//---------------------------------------------------------------------------------------------------------------
//
//  HAUD 2024.11.21
//
//
//  fb_Instance
//  - base class for process instance to work with fb_ProcessCollector
//  - basic check and var names, so you can build your procedures with it
//  - processes are connected via linked list
//
//  - inherit this base class for your application, call Check() cyclic
//
//---------------------------------------------------------------------------------------------------------------//
// This SOFTWARE is provided as an Exemple by THE PROVIDER "as is" and "with all faults." THE PROVIDER makes no  //
// representations or warranties of any kind concerning the safety, suitability, lack of viruses, inaccuracies,  //
// typographical errors, or other harmful components of this SOFTWARE. There are inherent dangers in the use of  //
// any software, and you are solely responsible for determining whether this SOFTWARE is compatible with your    //
// equipment and other software installed on your equipment. You are also solely responsible for the protection  //
// of your equipment and backup of your data, and THE PROVIDER will not be liable for any damages you may suffer //
// in connection with using, modifying, or distributing this SOFTWARE.                                           //
//---------------------------------------------------------------------------------------------------------------//
FUNCTION_BLOCK fb_Instance
VAR
  _eState                 : E_INSTANCE_STATE;  // local state machine for infeed procedure
  _eStateProgress         : E_PROGRESS; // substate for lacal state machine

  _eInit                  : E_PROGRESS;
  _eCheck                 : E_INSTANCE_CHECK;  // pointer checks

  // XTS station range
  _nStationLast           : UINT;
  _nStationFirst          : UINT;

  // process index
  _nProcess               : UINT;

  // local ctrl / state datafields for you to use
  _Ctrl                   : ST_PROCESS_CTRL;   // control to write, connected by reference to _ItfProcessCollector
  _State                  : ST_PROCESS_STATE;  // state   to read,  connected by reference to _ItfProcessCollector

  _ItfProcessCollector    : ARRAY[1..MAX_PROCESS] OF I_ProcessCollector;

  _ItfProcessList         : ARRAY[1..MAX_PROCESS] OF I_Process_LinkedList;  // access to all linked lists for process entry
  _ListResult             : ST_PROCESS_LIST_RESULT;
  _ProcessData            : ST_PROCESS_DATA;

  {attribute 'displaymode':='bin'}
  _wTargetUsed            : T_PROCESS;  // bits use XtsStation in target process
  _wTargetMask            : ARRAY[1..SIZEOF(T_PROCESS)*8] OF BYTE;

  _stMsg                  : ST_Message;
  _MessageLevel           : E_MessageType;
END_VAR

METHOD Check : BOOL // call this method in the extending/inheriting class
//-----------------------------------------------------------------------------
//-----------------------------------------------------------------------------
// plausibility checks
//-----------------------------------------------------------------------------
IF NOT (_nProcess > 0)
THEN
  _eCheck                 := E_INSTANCE_CHECK.INVALID_PROCESS_ID_ZERO;
  RETURN;
END_IF

IF NOT (_nProcess < MAX_PROCESS+1)
THEN
  _eCheck                 := E_INSTANCE_CHECK.INVALID_PROCESS_ID_MAX;
  RETURN;
END_IF
//-----------------------------------------------------------------------------
//-----------------------------------------------------------------------------
// pointer checks
//-----------------------------------------------------------------------------
IF NOT (_ItfProcessCollector[_nProcess] <> 0) 
THEN
  _eCheck                 := E_INSTANCE_CHECK.INVALID_INTERFACE_POINTER;
  RETURN;
END_IF

IF NOT (_ItfProcessCollector[_nProcess].ProcessId > 0)
THEN
  _eCheck                 := E_INSTANCE_CHECK.INVALID_PROCESS_ID_ZERO;
  RETURN;
END_IF

IF NOT (_ItfProcessCollector[_nProcess].ProcessId < MAX_PROCESS+1)
THEN
  _eCheck                 := E_INSTANCE_CHECK.INVALID_PROCESS_ID_MAX;
  RETURN;
END_IF

IF NOT (_nProcess = _ItfProcessCollector[_nProcess].ProcessId)
THEN
  _eCheck                 := E_INSTANCE_CHECK.INVALID_PROCESS_ID_NOTEQUAL_COLLECTOR_ID;
  RETURN;
END_IF

IF NOT (_ItfProcessList[_nProcess] <> 0)
THEN
  _eCheck                 := E_INSTANCE_CHECK.INVALID_INDEX_IN_LIST;
  RETURN;
END_IF
//-----------------------------------------------------------------------------
//-----------------------------------------------------------------------------
// connect datafields to interface of ProcessCollector
//-----------------------------------------------------------------------------
_ItfProcessCollector[_nProcess].ProcessCtrl      REF= _Ctrl;
_ItfProcessCollector[_nProcess].ProcessState     REF= _State;
//-----------------------------------------------------------------------------
//-----------------------------------------------------------------------------
// DEBUG: copy station range
//-----------------------------------------------------------------------------
_nStationLast                         := _ItfProcessCollector[_nProcess].StationLast;
_nStationFirst                        := _ItfProcessCollector[_nProcess].StationFirst;
//-----------------------------------------------------------------------------
//-----------------------------------------------------------------------------
// set message device
//-----------------------------------------------------------------------------
_stMsg.eDevice                        := e_Device.Process + _nProcess;
//-----------------------------------------------------------------------------
//-----------------------------------------------------------------------------
_eCheck                   := E_INSTANCE_CHECK.CHECK_DONE;
Check                     := TRUE;
END_METHOD

PROPERTY ProcessId : uint
GET
ProcessId := _nProcess;
END_GET
SET
_nProcess := ProcessId;
END_SET
END_PROPERTY

PROPERTY ProcessInterface : array[1..MAX_PROCESS] of I_ProcessCollector
SET
_ItfProcessCollector := ProcessInterface;
END_SET
END_PROPERTY

PROPERTY ProcessLinkedLists : ARRAY[1..max_process] OF I_Process_LinkedList
SET
_ItfProcessList := ProcessLinkedLists;
END_SET
END_PROPERTY

PROPERTY TargetUsed : T_PROCESS
GET
TargetUsed := _wTargetUsed;
END_GET
SET
_wTargetUsed := TargetUsed;
END_SET
END_PROPERTY

END_FUNCTION_BLOCK

(* stored: Version 1.1.0.1, ProductVersion 3.1.4024.13
   POU fb_Instance: Id {02367fcb-67b8-497b-8382-1c3639f01a80}, SpecialFunc None
   Folder properties: Id {5f969983-7274-474e-ad53-ecf15d94990d}
   Method Check: Id {04192027-e492-4023-92ca-671af767f088}
   Property ProcessId: Id {bc02b386-af4a-427a-bfae-f03f977e543e}
   Get Get: Id {f26a4457-27eb-4b2a-bb3e-26741e3e8a80}
   Set Set: Id {82f5dac8-30d1-408a-8463-5b7d3dbc951d}
   Property ProcessInterface: Id {7856fb23-1ef1-472e-9855-7bec6a7c2039}
   Set Set: Id {d83e93f2-0907-4e4e-899d-c33bd6f05c59}
   Property ProcessLinkedLists: Id {f1f4c45b-0247-4e47-9cfc-0c8d3318a647}
   Set Set: Id {d5137f63-8b56-4b2c-a086-29d9076bed68}
   Property TargetUsed: Id {2b5cddab-4380-4158-b4c4-d19cd4b73a48}
   Get Get: Id {badbc8e4-3616-4206-9b21-715f9daff180}
   Set Set: Id {8caea5fe-4a35-426a-aec0-99973bf00216} *)
